// TIA Portal V20 export
// export: Created 2025-12-01T14:57:07.0563262Z, ExportSetting None, DisplayName Totally Integrated Automation Portal, DisplayVersion V20 Update 3, DisplayName TIA Portal Openness, DisplayVersion V20 Update 3, DisplayName TIA Portal Version Control Interface, DisplayVersion V20 Update 3, DisplayName STEP 7 Professional, DisplayVersion V20 Update 3, DisplayName STEP 7 Safety, DisplayVersion V20 Update 2, DisplayName WinCC Basic/Comfort/Advanced, DisplayVersion V20 Update 3, DisplayName WinCC Professional, DisplayVersion V20 Update 3, DisplayName WinCC Unified, DisplayVersion V20 Update 3
FUNCTION "FC989_CTRL_VAR_MOVIMOT_ASi" : Void   // FC989, SCL
{ S7_Optimized_Access := 'FALSE' }
VERSION : 0.0
// Parámetros del bloque
// stored: AutoNumber false, SetENOAutomatically false
   VAR_INPUT
      Dir_LineaGW : Int;
      Num_Slave : Int;
      Avanzar : Bool;
      Retroceder : Bool;
      Velocidad : Int;
      Inversion : Bool;
      Rearme : Bool;
   END_VAR
   VAR_OUTPUT
      En_Movimiento : Bool;
      Error : Bool;
      NumEnvio : Int;
   END_VAR
   VAR_TEMP
      Codigo : Int;
      CW AT Codigo : Struct
         high_0 : Bool;
         high_1 : Bool;
         high_2 : Bool;
         high_3 : Bool;
         high_4 : Bool;
         high_5 : Bool;
         high_6 : Bool;
         high_7 : Bool;
         BitVel_0 : Bool;
         BitVel_1 : Bool;
         BitVel_2 : Bool;
         BitVel_3 : Bool;
         low_4 : Bool;
         low_5 : Bool;
         low_6 : Bool;
         low_7 : Bool;
      END_STRUCT;
      Offset_Byte : Int;
      Offset_Bit : Int;
   END_VAR
BEGIN


       // Área de instrucciones
       //Las cabeceras ASI están dentro de la imagen de proceso, por lo que accedemos directamente

       #Offset_Bit := 4 - ((#Num_Slave MOD 2)*4) ;
       #Offset_Byte := ((#Num_Slave + 1) / 2 ) - (#Num_Slave MOD 2);

       (* classic code: #En_Movimiento := %EX((#Dir_LineaGW + #Offset_Byte), (0 + #Offset_Bit));*)
       #En_Movimiento := PEEK_BOOL(area:=16#81,dbNumber:=0,byteOffset:=(#Dir_LineaGW + #Offset_Byte),bitOffset:=(0 + #Offset_Bit));
       (* classic code: #Error := %EX((#Dir_LineaGW + #Offset_Byte), (1 + #Offset_Bit));*)
       #Error := PEEK_BOOL(area:=16#81,dbNumber:=0,byteOffset:=(#Dir_LineaGW + #Offset_Byte),bitOffset:=(1 + #Offset_Bit));

       IF #Avanzar AND NOT #Retroceder AND NOT #Error AND #Velocidad <> 0 THEN
           // Área de instrucciones_IF
           IF NOT #Inversion THEN 
               IF #Velocidad > 7 THEN #Codigo := 13;
               ELSE     #Codigo := (#Velocidad * 2) - 1; 
               END_IF;
           ELSE
               IF #Velocidad > 7 THEN #Codigo := 14;
               ELSE #Codigo := #Velocidad * 2;
               END_IF;
           END_IF;

       ELSIF NOT #Avanzar AND #Retroceder AND NOT #Error AND #Velocidad <> 0 THEN
           // Área de instrucciones_ELSIF
           IF #Inversion THEN 
               IF #Velocidad > 7 THEN #Codigo := 13;
               ELSE     #Codigo := (#Velocidad * 2) - 1; 
               END_IF;
           ELSE
               IF #Velocidad > 7 THEN #Codigo := 14;
               ELSE #Codigo := #Velocidad * 2;
               END_IF;
           END_IF;

       ELSIF #Error AND #Rearme THEN
           // Área de instrucciones_ELSIF
           #Codigo := 15;
       ELSE
           // Área de instrucciones_ELSE
           #Codigo := 0;
       END_IF;

       #NumEnvio := #Codigo ;
       //Las cabeceras ASI están dentro de la imagen de proceso, por lo que accedemos directamente
       (* classic code: %AX((#Dir_LineaGW + #Offset_Byte), (0 + #Offset_Bit)) := #CW.BitVel_0;*)
       POKE_BOOL(area:=16#82,dbNumber:=0,byteOffset:=(#Dir_LineaGW + #Offset_Byte),bitOffset:=(0 + #Offset_Bit),value:=#CW.BitVel_0)  ;
       (* classic code: %AX((#Dir_LineaGW + #Offset_Byte), (1 + #Offset_Bit)) := #CW.BitVel_1;*)
       POKE_BOOL(area:=16#82,dbNumber:=0,byteOffset:=(#Dir_LineaGW + #Offset_Byte),bitOffset:=(1 + #Offset_Bit),value:=#CW.BitVel_1)  ;
       (* classic code: %AX((#Dir_LineaGW + #Offset_Byte), (2 + #Offset_Bit)) := #CW.BitVel_2;*)
       POKE_BOOL(area:=16#82,dbNumber:=0,byteOffset:=(#Dir_LineaGW + #Offset_Byte),bitOffset:=(2 + #Offset_Bit),value:=#CW.BitVel_2)  ;
       (* classic code: %AX((#Dir_LineaGW + #Offset_Byte), (3 + #Offset_Bit)) := #CW.BitVel_3;*)
       POKE_BOOL(area:=16#82,dbNumber:=0,byteOffset:=(#Dir_LineaGW + #Offset_Byte),bitOffset:=(3 + #Offset_Bit),value:=#CW.BitVel_3)  ;
END_FUNCTION
